TYPE E_ITC_FunctionControlCode :
(**************************************************************************************
 * 	Application		:	BoxControl Framework
 *	Revision		:	$Revision: 404529 $
 *	Revision date	:	$Date: 2018-04-23 08:21:38 +0200 (Mo., 23 Apr 2018) $
 *	Last changed by	:	$Author: b7bolm $
 *	URL				:	$URL: http://almscdc.swisslog.com/repo/SWPD/Development/BoxControlFramework/20_Release/trunk/01_Software/BCF/BCF/JumpStart/20_Product/10_App/12_E_Functions/10_Lib/10_Conv/01_DUTs/E_ITC_FunctionControlCode.TcDUT $
 *
 *	Purpose			:	Element function control request code
 *
 * ------------------------------------------------------------------------------------
 *	Copyright Swisslog [IP AG], Switzerland. All rights reserved.
 * 
 * ------------------------------------------------------------------------------------
 *	
 * 	Revision History: 
 *
 * 	VERSION			DATE			INITIALS			DESCRIPTION
 *	0.1				01.01.2001		swl					Example
 *
 **************************************************************************************)
(
	NO_CODE					:= 0, // No code
	RESET_ERROR 			:= 1, // Reset Error
	INITIALIZE 				:= 2, // Initialize
	ENABLE 					:= 4, // Enable / Disable
	SET_VARIABLE 			:= 5, // Set Variable
	SET_ERROR 				:= 20 // Set Error
);
END_TYPE

(* stored: Version 1.1.0.1, ProductVersion 3.1.4022.12
   DUT E_ITC_FunctionControlCode: Id {864faf8e-9ebb-47b3-8603-9933d3d4fd57} *)
